(* IEC 61131-3 sources: YaoKangDeviceDemo/src, 1 file *)

(* ---- PRG_Main.st ---- *)
(*============================================================================
  PRG_Main —— 主扫描（唯一任务入口，固定调用链，顺序不可调整）
  ----------------------------------------------------------------------------
  扫描链（开发计划 P1）：
    1  PRG_CmdPreclear    命令残留清理（脉冲边沿方案后主要兜底电平离态）
    2  PRG_InputAdapter   I/O 镜像去抖 + HMI 命令解析（R_TRIG 脉冲/电平）
    3  PRG_Monitor        AD/传感器采集与 plausibility 诊断
    4  PRG_ErrorManager   错误唯一写入：活动错误/警告/历史队列
    5  PRG_SafetyManager  安全独立常驻：急停链/防夹/超力/堵转/限位
    6  PRG_ModeManager    系统状态机：iState 唯一写入（13 态仲裁）
    7  PRG_TaskRunner     任务分派：AUTORUN/SELFTEST/HOMING/CALIBRATE/RESET
    8  PRG_ParamService   参数三区 + ConfigCmd + 设备身份（P5/P11）
    9  PRG_Power          伺服上下电分时管理：轴使能唯一写入
    10 PRG_OutputAdapter  执行器 + MC 指令唯一调用点（3×M900 / 推杆）
    11 PRG_HmiOutput      内部状态 → D 区回填（最末环，不碰命令位）

  单写源：每个对外变量唯一写入者，见各程序头注释。
  HMI 映射：HMI AT %MW200（Stru_HMI）、HMI_DeviceIdentity AT %MW1000、
            HMI_DeviceIdentityWrite AT %MW1010（见 GVL_HMI.st）。
==========================================================================*)
PROGRAM PRG_Main
VAR
    (* H5U 定时器为内联指令 TONR(IN:=,PT:=,Q=>布尔位)，无需 TON 实例；
       tScanWatchdog 即看门狗 TONR 的 Q=> 输出 BOOL（超时置位）。 *)
    tScanWatchdog   : BOOL;   (* 扫描看门狗超时标志（Q=>tScanWatchdog） *)
END_VAR

(*--- 扫描看门狗（周期以任务组态为准，超时交 SAFETY/ERROR 处理） ---*)
TONR(IN := TRUE, PT := T#50MS, Q => tScanWatchdog);

(*--- 固定扫描链 ---*)
PRG_CmdPreclear();
PRG_InputAdapter();
PRG_Monitor();
PRG_ErrorManager();
PRG_SafetyManager();
PRG_ModeManager();
PRG_TaskRunner();
PRG_ParamService();
PRG_Power();
PRG_OutputAdapter();
PRG_HmiOutput();
END_PROGRAM
